FUNCTION_BLOCK T_ModeInitialisedFromInvalidToProduction EXTENDS T_UnitTestBase
VAR
  mockState : T_MockStateModule;
  modeManager : T_ModeManager(mockState);
  expected, actual : UINT;
END_VAR

CycleModuleLogicToAllowChangesToFilterThrough();

expected := TO_UINT(E_PMLUnitMode.ePMLUnitMode_Production);
actual := TO_UINT(modeManager._CurrentMode);
assertion.AssertEquals_UINT(expected, actual, 'actual := modeManager._CurrentMode'); 

TestFinished();

METHOD CycleModuleLogicToAllowChangesToFilterThrough : BOOL
VAR_INST
	i: INT;

END_VAR
modeManager.CyclicLogic();
CycleModuleLogicToAllowChangesToFilterThrough := i >= 10;
i := SEL(i >= 10, i + 1, 0);
END_METHOD

END_FUNCTION_BLOCK

(* stored: Version 1.1.0.1, ProductVersion 3.1.4024.12
   POU T_ModeInitialisedFromInvalidToProduction: Id {7a8b6319-64c3-428e-a95a-938b00277ced}, SpecialFunc None
   Method CycleModuleLogicToAllowChangesToFilterThrough: Id {dbbabcf2-0662-4caf-9f32-66a817ad1d97} *)
